FUNCTION_BLOCK FB_STATION
VAR_INPUT
	eSTATE:E_STATE:=E_STATE.uninit;
	sSTATION_STATE:STRING:='UNINIT';
	sName:STRING;
	bHOMED : BOOL:=FALSE;
	tACTION:TON;
	bPAUSE:BOOL:=FALSE;
	
END_VAR
VAR_OUTPUT
END_VAR
VAR
	
	bRESET:BOOL;
	bSTART:BOOL:=FALSE;
	iSTATION_STATE:INT:=98;;
	bFIRST_RUB:BOOL:=FALSE;
END_VAR

END_FUNCTION_BLOCK

(* stored: Version 1.1.0.1, ProductVersion 3.1.4024.12
   POU FB_STATION: Id {af24db28-040e-471c-ad69-35306a54a2e6}, SpecialFunc None *)
